(* CODESYS project Integracao_Python_Codesys_OPCUA.project

Project tree, tasks and I/O mapping:
  Device : CODESYS Control Win V3, 3S - Smart Software Solutions GmbH, order no. 305021, version 3.5.11.30
    DeviceApplication
      application Application
        libraries: Standard, * (System)
        task MainTask (cyclic, interval t#20ms, priority 1) calls PLC_PRG
        program PLC_PRG [LD]
        global variables GVL
        Symbols
*)

// Device/DeviceApplication/Application/GVL
{attribute 'qualified_only'}
VAR_GLOBAL
	//ENTRADAS
	DETECTA_VERMELHO, DETECTA_VERDE:BOOL;
	//SAIDAS
	ATUADOR_VERMELHO,ATUADOR_VERDE:BOOL;
END_VAR

// Device/DeviceApplication/Application/PLC_PRG
PROGRAM PLC_PRG
VAR
END_VAR

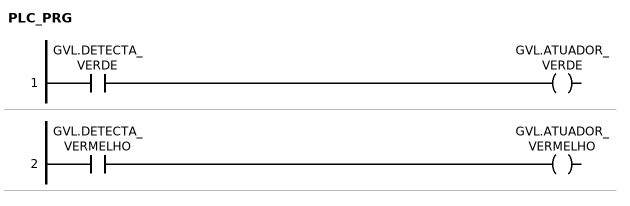
// NETWORK 1
GVL.ATUADOR_VERDE := GVL.DETECTA_VERDE;

// NETWORK 2
GVL.ATUADOR_VERMELHO := GVL.DETECTA_VERMELHO;

END_PROGRAM
